FUNCTION_BLOCK RunInitScaraAndRack EXTENDS RunUnitGeneric
VAR_INPUT
	scara : POINTER TO RunScaraAgent;
	racks : ARRAY[0..1] OF POINTER TO RunCommonRack;
	bridges : ARRAY[0..3] OF POINTER TO RunBridge;
END_VAR
VAR_OUTPUT
END_VAR
VAR
	nCounter : INT;
END_VAR

SUPER^();



CASE outputState OF 
	eSpecialStates.INITIAL_BEGIN:
		bSerialTransition := scara^.Initialize();
	eSpecialStates.INITIAL_STATE_1:
		bSerialTransition := TRUE;
		FOR nCounter:=0 TO 1 BY 1 DO
			bSerialTransition := bSerialTransition AND racks[nCounter]^.Initialize();
		END_FOR
	eSpecialStates.INITIAL_STATE_2:
		bSerialTransition := TRUE;
		FOR nCounter:=0 TO 3 BY 1 DO
			IF bridges[nCounter]<>0 THEN
				bSerialTransition := bSerialTransition AND bridges[nCounter]^.Initialize();
			END_IF	
		END_FOR
		IF bSerialTransition THEN
			NextState := eSpecialStates.INITIAL_END; //ready for action
		END_IF
	//---------------------
	//	Then start working
	//---------------------
	eSpecialStates.GENERIC_GROUP_START:
		scara^.NextState := eSpecialStates.GENERIC_GROUP_START; //start working
		FOR nCounter:=0 TO 1 BY 1 DO
			racks[nCounter]^.NextState := eSpecialStates.GENERIC_GROUP_START;
		END_FOR
		FOR nCounter:=0 TO 3 BY 1 DO
			IF bridges[nCounter]<>0 THEN
				bridges[nCounter]^.NextState := eSpecialStates.GENERIC_GROUP_START;
			END_IF	
		END_FOR
		bSerialTransition := TRUE; // to void state
END_CASE

END_FUNCTION_BLOCK

(* stored: Version 1.1.0.1, ProductVersion 3.1.4024.0
   POU RunInitScaraAndRack: Id {152d0302-1d9a-4db0-acac-27fa8a45876a}, SpecialFunc None *)
